Fanuc TP program (LS listing): OPEN_T2.LS

/PROG  OPEN_T2	  Macro
/ATTR
OWNER		= MNEDITOR;
COMMENT		= "";
PROG_SIZE	= 216;
CREATE		= DATE 25-07-07  TIME 18:39:38;
MODIFIED	= DATE 25-07-07  TIME 19:13:16;
FILE_NAME	= GRIPPER_;
VERSION		= 0;
LINE_COUNT	= 2;
MEMORY_SIZE	= 580;
PROTECT		= READ_WRITE;
TCD:  STACK_SIZE	= 0,
      TASK_PRIORITY	= 50,
      TIME_SLICE	= 0,
      BUSY_LAMP_OFF	= 0,
      ABORT_REQUEST	= 0,
      PAUSE_REQUEST	= 0;
DEFAULT_GROUP	= *,*,*,*,*;
CONTROL_CODE	= 00000000 00000000;
/APPL
/MN
   1:  RO[1:ON :open T2]=ON ;
   2:  //RO[2:OFF:close T2]=OFF ;
/POS
/END
